// TIA Portal V20 export
TYPE "Fault"
// stored: Access Published, Namespace LineA1
   STRUCT
      Motor_Error : Bool;
      Sensor_Blockage : Bool;
   END_STRUCT;
END_TYPE
